// TIA Portal V16 export
// export: Created 2024-05-10T06:46:43.8068816Z, ExportSetting WithDefaults, DisplayName Totally Integrated Automation Portal, DisplayVersion V16, DisplayName TIA Portal Version Control Interface, DisplayVersion V16, DisplayName TIA Portal Openness, DisplayVersion V16, DisplayName STEP 7 Professional, DisplayVersion V16, DisplayName STEP 7 Safety, DisplayVersion V16, DisplayName WinCC Professional, DisplayVersion V16
DATA_BLOCK "K21_ST09上自动_DB"   // DB21
VERSION : 0.1
// stored: AutoNumber false, DBAccessibleFromOPCUA true, InstanceOfName K21_ST09上自动, InstanceOfType FB
"K21_ST09上自动"
BEGIN
END_DATA_BLOCK
